// TIA Portal V19 export
VAR_GLOBAL   // PLC tag table "D14"
   D14_Lp_EntryReq_LB203 AT %Q109.2 : Bool;   // 240SH1
   D14_Lp_SafetyReset_LB203 AT %Q109.3 : Bool;   // 240SH2
   D14_Pb_EntryReq_LB203 AT %I108.0 : Bool;   // 240SH1
   D14_Pb_SafetyReset_LB203 AT %I108.1 : Bool;   // 240SH2
   D14_Comando_Elettroserratura AT %Q109.1 : Bool;   // 24002
   D14_Cancello_Chiuso AT %I107.6 : Bool;   // 24001
   D14_Cancello_Bloccato AT %I107.7 : Bool;   // 24003
   D14_Ls_Os1 AT %I1079.1 : Bool;   // 106DI1 - 240A1
   D14_Ls_Os2 AT %I1079.5 : Bool;   // 106DI5 - 240A1
END_VAR
